# EPICS autosave request: TLBC2App/Db/ADTLBC2_settings.req
file "ADBase_settings.req", P=$(P), R=$(R)
$(P)$(R)Attenuation
$(P)$(R)AutoCalcAreaClipLevel
$(P)$(R)AutoExposure
$(P)$(R)Wavelength
